FUNCTION_BLOCK BINARY_TO_DEC
VAR_INPUT
	BIN0 : BOOL; //Bemenet MSB
	BIN1 : BOOL; //Bemenet
	BIN2 : BOOL; //Bemenet 
END_VAR
VAR_OUTPUT
	ID : INT; // kimeneti int
	
END_VAR
VAR
	bH : ARRAY [0..2] OF  INT; // helyiértékek értékei
	i : UINT;
END_VAR


FOR i :=0 TO 2 DO
	bH[i] :=(LREAL_TO_INT( EXPT(2,i)));
	
END_FOR
ID := (BOOL_TO_INT(BIN0)* bH[0])+ BOOL_TO_INT(BIN1)*bH[1]+BOOL_TO_INT(BIN2)*bH[2];

END_FUNCTION_BLOCK

(* stored: Version 1.1.0.1, ProductVersion 3.1.4024.11
   POU BINARY_TO_DEC: Id {020b1aef-5911-45e8-82a8-d58a78ccd987}, SpecialFunc None *)
